FUNCTION_BLOCK MUL_UINT (* IEC 61131-3 UINT Multiplication *)
  (* Standard: 61131-3 *)
  (* Version 0.0, 2004-12-15, JHC, Rockwell Automation, Converted from SRC format. *)
  (* Compiler header: package fb.rt.plc.math; *)
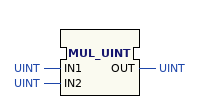
  VAR_INPUT
    IN1 : UINT; (* Multiplicand *)
    IN2 : UINT; (* Multiplier *)
  END_VAR
  VAR_OUTPUT
    OUT : UINT; (* Product *)
  END_VAR
END_FUNCTION_BLOCK
